TYPE ST_UnwindRecipe :
    STRUCT
        Axis : ST_AxisRecipe;
    END_STRUCT
END_TYPE

(* stored: Version 1.1.0.1
   DUT ST_UnwindRecipe: Id {735d15fd-3b33-4998-bd22-58278c0a1fb4} *)
